// TIA Portal V17 export
// export: Created 2024-08-07T21:44:05.8548651Z, ExportSetting WithDefaults, DisplayName Totally Integrated Automation Portal, DisplayVersion V17 Update 7, DisplayName TIA Portal Openness, DisplayVersion V17 Update 7, DisplayName TIA Portal Version Control Interface, DisplayVersion V17, DisplayName SINAMICS Startdrive Advanced, DisplayVersion V17 SP2, DisplayName SINAMICS Startdrive G110M, G120, G120C, G120D, G120P, G115D, DisplayVersion V17 SP2, DisplayName SINAMICS Startdrive G130, G150, S120, S150, SINAMICS MV, S210, DisplayVersion V17 SP2, DisplayName STEP 7 Professional, DisplayVersion V17 Update 7, DisplayName STEP 7 Safety, DisplayVersion V17 Update 6, DisplayName WinCC Advanced / Unified PC, DisplayVersion V17 Update 7
DATA_BLOCK "HMIData"   // DB1
{ S7_Optimized_Access := 'TRUE' }
VERSION : 0.1
// stored: AutoNumber false, DBAccessibleFromOPCUA true, DBAccessibleFromWebserver true, IsOnlyStoredInLoadMemory false, IsRetainMemResEnabled false, IsWriteProtectedInAS false, MemoryReserve 100
   VAR
      HMI { S7_SetPoint := 'True'} : "UDT_HMI";
      ManualCommandHMI : Int := 0;
      ManualCommand : Int := 0;
   END_VAR
BEGIN
   HMI.ScreenData[1..5] := 16#0000;
   HMI.UserNumber := 0;
   HMI.ActualScreenNumber := 0;
   HMI.RequiredScreenNumber := 0;
   HMI.FunctionKeys[1..8] := FALSE;
END_DATA_BLOCK
